{attribute 'qualified_only'}
{attribute 'strict'}
{attribute 'to_string'}
TYPE E_Interlock :
(
	AlarmTrig,
	WarningTrig,
	N2PressureLowAlarm,
	N2PressureLowWaring,
	H2PressureLowAlarm,
	H2PressureLowWarning,
	NH3PressureLowAlarm,
	NH2PressureLowWaring,
	SiH4PressureLowAlarm,
	SiH4PressureLowWarning,
	RecipeStartEnable,
	ReactorOpenEnable,
	HeatercanbeturnON,
	PumpcanbeturnON,  // GVL_IO.aInterlock[1].13
	
	ALARM_POPUP_GasPressureLowN2,
	ALARM_POPUP_GasPressureLowH2,
	ALARM_POPUP_GasPressureLowNH3,
	ALARM_POPUP_GasPressureLowSiH4,
	ALARM_POPUP_CWTemperatureHighSH,
	ALARM_POPUP_CWTemperatureHighCoil,
	ALARM_POPUP_SusceptorOverTemperature,
	ALARM_POPUP_ReactorOverPressure,
	ALARM_POPUP_PneumaticPressureLow,
	ALARM_POPUP_CoolingWaterLow,
	ALARM_POPUP_InductionHeaterFault,
	ALARM_POPUP_RotationMotorFault,
	ALARM_POPUP_VacuumPumpFault,
	ALARM_POPUP_GasCabinetDoorOpen,
	ALARM_POPUP_ReactorCabinetDoorOpen,
	ALARM_POPUP_SusceptorTemperatureDeviation,
	ALARM_POPUP_ReactorPressureDeviation,
	ALARM_POPUP_SusceptorRotationDeviation,
	ALARM_POPUP_MORunDeviation,
	ALARM_POPUP_HydRunDeviation,
	ALARM_POPUP_NH3LargeINDeviation,
	ALARM_POPUP_NH3SmallINDeviation,
	ALARM_POPUP_SiHINDeviation,
	ALARM_POPUP_SiHDilutionDeviation,
	ALARM_POPUP_SiHDilutedDeviation,
	ALARM_POPUP_TEBBubblingDeviation,
	ALARM_POPUP_TMAlBubblingDeviation,
	ALARM_POPUP_TMInBubblingDeviation,
	ALARM_POPUP_TMGaBubblingDeviation,
	ALARM_POPUP_DTMGaBubblingDeviation,
	ALARM_POPUP_DTMGaDilutionDeviation,
	ALARM_POPUP_DTMGaDilutedDeviation,
	ALARM_POPUP_Cp2MgBubblingDeviation,
	ALARM_POPUP_ReactorPurgeDeviation,
	ALARM_POPUP_RotationSealPurgeDeviation,
	ALARM_POPUP_MOVentDeviation,
	ALARM_POPUP_HydVentDeviation,
	ALARM_POPUP_SiH4PressureDeviation,
	ALARM_POPUP_TEBPressureDeviation,
	ALARM_POPUP_TMAlPressureDeviation,
	ALARM_POPUP_TMInPressureDeviation,
	ALARM_POPUP_TMGaPressureDeviation,
	ALARM_POPUP_DTMGaPressureDeviation,
	ALARM_POPUP_Cp2MgPressureDeviation,
	WARNING_POPUP_GasPressureLowN2,
	WARNING_POPUP_GasPressureLowH2,
	WARNING_POPUP_GasPressureLowNH3,
	WARNING_POPUP_GasPressureLowSiH4,
	WARNING_POPUP_CWTemperatureHighSH,
	WARNING_POPUP_CWTemperatureHighCoil,
	WARNING_POPUP_SusceptorOverTemperature,
	WARNING_POPUP_ReactorOverPressure,
	WARNING_POPUP_PneumaticPressureLow,
	WARNING_POPUP_CoolingWaterLow,
	WARNING_POPUP_InductionHeaterFault,
	WARNING_POPUP_RotationMotorFault,
	WARNING_POPUP_VacuumPumpFault,
	WARNING_POPUP_GasCabinetDoorOpen,
	WARNING_POPUP_ReactorCabinetDoorOpen,
	WARNING_POPUP_SusceptorTemperatureDeviation,
	WARNING_POPUP_ReactorPressureDeviation,
	WARNING_POPUP_SusceptorRotationDeviation,
	WARNING_POPUP_MORunDeviation,
	WARNING_POPUP_HydRunDeviation,
	WARNING_POPUP_NH3LargeINDeviation,
	WARNING_POPUP_NH3SmallINDeviation,
	WARNING_POPUP_SiHINDeviation,
	WARNING_POPUP_SiHDilutionDeviation,
	WARNING_POPUP_SiHDilutedDeviation,
	WARNING_POPUP_TEBBubblingDeviation,
	WARNING_POPUP_TMAlBubblingDeviation,
	WARNING_POPUP_TMInBubblingDeviation,
	WARNING_POPUP_TMGaBubblingDeviation,
	WARNING_POPUP_DTMGaBubblingDeviation,
	WARNING_POPUP_DTMGaDilutionDeviation,
	WARNING_POPUP_DTMGaDilutedDeviation,
	WARNING_POPUP_Cp2MgBubblingDeviation,
	WARNING_POPUP_ReactorPurgeDeviation,
	WARNING_POPUP_RotationSealPurgeDeviation,
	WARNING_POPUP_MOVentDeviation,
	WARNING_POPUP_HydVentDeviation,
	WARNING_POPUP_SiH4PressureDeviation,
	WARNING_POPUP_TEBPressureDeviation,
	WARNING_POPUP_TMAlPressureDeviation,
	WARNING_POPUP_TMInPressureDeviation,
	WARNING_POPUP_TMGaPressureDeviation,
	WARNING_POPUP_DTMGaPressureDeviation,
	WARNING_POPUP_Cp2MgPressureDeviation,
	E_Interlock_END
);
END_TYPE

(* stored: Version 1.1.0.1
   DUT E_Interlock: Id {6f0be869-79f2-4c6e-a450-409068652e13} *)
